{attribute 'qualified_only'}
VAR_GLOBAL
	//VoltMonDB : ARRAY [1..2] OF ST_VoltMon_Base; 
END_VAR

(* stored: Version 1.1.0.1, ProductVersion 3.1.4024.11
   GVL VoltMonitor_DB: Id {860f77a6-4bc2-402b-92d3-cf7c77cd35cf} *)
